{attribute addProperty BoxType "KL9999"}
{attribute addProperty Id "VarInAT %I*UINT000VarOutAT %Q*UINT000"}
{attribute addProperty CRC "573873137"}
{attribute addProperty SizeInBites "0"}
{attribute addProperty SizeInBytes "0"}
TYPE Channel_22349BF1 :
STRUCT
	{attribute addProperty Name "VarIn"}
	VarIn AT %I* : UINT;
	{attribute addProperty Name "VarOut"}
	VarOut AT %Q* : UINT;
END_STRUCT
END_TYPE

(* stored: Version 1.2.0.0, ProductVersion 3.1.4024.9
   DUT Channel_22349BF1: Id {ce8e987e-4d9f-4c5a-a271-891f83879a96} *)
